//----------------------------------------------------------------------------//
//            Copyright 2018 Rieckermann Engineering Operations               //
//----------------------------------------------------------------------------//
// Class:       fbTC1                                                         //
// Description:                                                               //
// Cooling only temperature controller.                                       //
//----------------------------------------------------------------------------//
// Revision history:                                                          //
// Rev By               Date        CC        Note                            //
// 2.0 David Paspa      24-Apr-2018 NA        Reboot for S7-1500.             //
// 0.7 Gerald Kontriner 09-Oct-2009 CC-09/016 MON_MISMATCH Logic.             //
// 0.6 Khairul Basar    06-Oct-2009 CC-09/016 PID HLM,LLM reversed for cool.  //
// 0.5 Khairul Basar    17-Sep-2009 CC-09/016 OUT_CMD as Command to MOD1 added//
// 0.4 Khairul Basar    16-Sep-2009 CC-09/016 Duplicate Auto/man parameters   //
//                                            deleted auto/manual both now    //
//                                            using same parameters.          //
// 0.3 Khairul Basar    11-Sep-2009 CC-09/016 Manual setpoint, Non PID        //
//                                            selection parameters added &    //
//                                            programmed..                    //
// 0.2 Khairul Basar    03-Sep-2009 CC-09/016 State enable/disable code added //
//                                            NTERLOCK is changed from        //
//                                            IN_OUT to OUT & program safe    //
//                                            state for Interlock.            //
//                                            CMD_AUTO/MAN & DEV_STATE.       //
//                                            paramters are added & programed.//
// 0.1 Khairul Basar    03-Aug-2009           Initial design.                 //
//----------------------------------------------------------------------------//
FUNCTION_BLOCK "fbTC1"
TITLE = TC1 : Vesel cooling only temperature controller
{ S7_Optimized_Access := 'TRUE' }
AUTHOR : REO
NAME : fbTC1
VERSION : 2.0

//----------------------------------------------------------------------------//
// Declare interface and variables:                                           //
//----------------------------------------------------------------------------//
VAR
    p : "udtTC1";            // Block data interface
    PID1 {ReadalPartName := 'CONT_C'; LibVersion := '1.0'} : CONT_C;
END_VAR

VAR_TEMP
    cmdEnable : Bool;
    cmdDisable : Bool;
    tSetpoint : Real;
    tManual_Not_PID : Bool;
END_VAR

BEGIN
NETWORK
TITLE = Check if the TCV is not in AUTO and REMOTE
    //------------------------------------------------------------------------//
    // INTERLOCK   INTERLOCK   INTERLOCK   INTERLOCK   INTERLOCK   INTERLOCK  //
    // INTERLOCK   INTERLOCK   INTERLOCK   INTERLOCK   INTERLOCK   INTERLOCK  //
    //                                                                        //
    // Check if the TCV cannot be controlled if not in AUTO:                  //
    //------------------------------------------------------------------------//
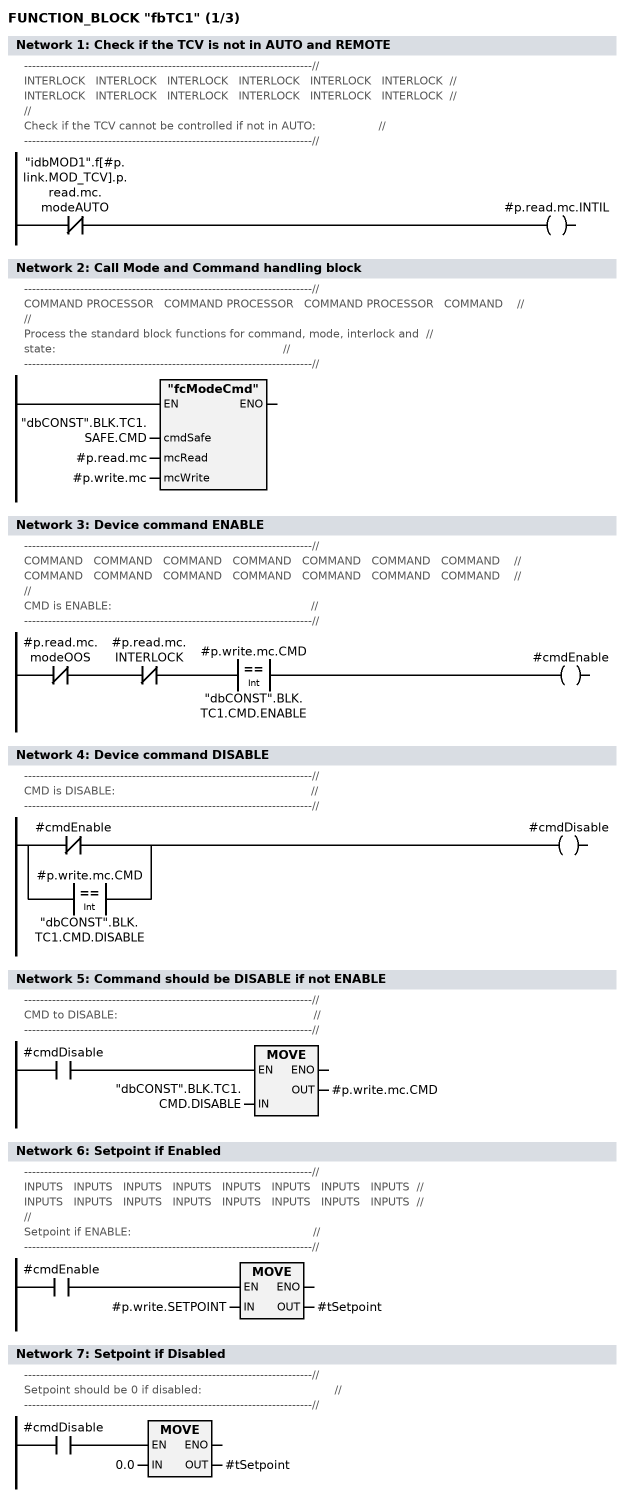
    AN "idbMOD1".f[#p.link.MOD_TCV].p.read.mc.modeAUTO;
    = #p.read.mc.INTIL;

NETWORK
TITLE = Call Mode and Command handling block
    //------------------------------------------------------------------------//
    // COMMAND PROCESSOR   COMMAND PROCESSOR   COMMAND PROCESSOR   COMMAND    //
    //                                                                        //
    // Process the standard block functions for command, mode, interlock and  //
    // state:                                                                 //
    //------------------------------------------------------------------------//
    CALL "fcModeCmd"
    (   cmdSafe              := "dbCONST".BLK.TC1.SAFE.CMD ,
        mcRead               := #p.read.mc ,
        mcWrite              := #p.write.mc
    );

NETWORK
TITLE = Device command ENABLE
    //------------------------------------------------------------------------//
    // COMMAND   COMMAND   COMMAND   COMMAND   COMMAND   COMMAND   COMMAND    //
    // COMMAND   COMMAND   COMMAND   COMMAND   COMMAND   COMMAND   COMMAND    //
    //                                                                        //
    // CMD is ENABLE:                                                         //
    //------------------------------------------------------------------------//
    AN #p.read.mc.modeOOS;
    AN #p.read.mc.INTERLOCK;
    A(;
    L #p.write.mc.CMD;
    L "dbCONST".BLK.TC1.CMD.ENABLE;
    ==I;
    );
    = #cmdEnable;

NETWORK
TITLE = Device command DISABLE
    //------------------------------------------------------------------------//
    // CMD is DISABLE:                                                        //
    //------------------------------------------------------------------------//
    ON #cmdEnable;
    O(;
    L #p.write.mc.CMD;
    L "dbCONST".BLK.TC1.CMD.DISABLE;
    ==I;
    );
    = #cmdDisable;

NETWORK
TITLE = Command should be DISABLE if not ENABLE
    //------------------------------------------------------------------------//
    // CMD to DISABLE:                                                        //
    //------------------------------------------------------------------------//
    A #cmdDisable;
    JCN _a;
    L "dbCONST".BLK.TC1.CMD.DISABLE;
    T #p.write.mc.CMD;
_a:   NOP 0;

NETWORK
TITLE = Setpoint if Enabled
    //------------------------------------------------------------------------//
    // INPUTS   INPUTS   INPUTS   INPUTS   INPUTS   INPUTS   INPUTS   INPUTS  //
    // INPUTS   INPUTS   INPUTS   INPUTS   INPUTS   INPUTS   INPUTS   INPUTS  //
    //                                                                        //
    // Setpoint if ENABLE:                                                    //
    //------------------------------------------------------------------------//
    A #cmdEnable;
    JCN _b;
    L #p.write.SETPOINT;
    T #tSetpoint;
_b:   NOP 0;

NETWORK
TITLE = Setpoint if Disabled
    //------------------------------------------------------------------------//
    // Setpoint should be 0 if disabled:                                      //
    //------------------------------------------------------------------------//
    A #cmdDisable;
    JCN _c;
    L 0.0;
    T #tSetpoint;
_c:   NOP 0;

NETWORK
TITLE = PID in manual if disabled or manual flag set
    //------------------------------------------------------------------------//
    // OUTPUTS   OUTPUTS   OUTPUTS   OUTPUTS   OUTPUTS   OUTPUTS   OUTPUTS    //
    // OUTPUTS   OUTPUTS   OUTPUTS   OUTPUTS   OUTPUTS   OUTPUTS   OUTPUTS    //
    //                                                                        //
    // PID in manual mode if requested:                                       //
    //------------------------------------------------------------------------//
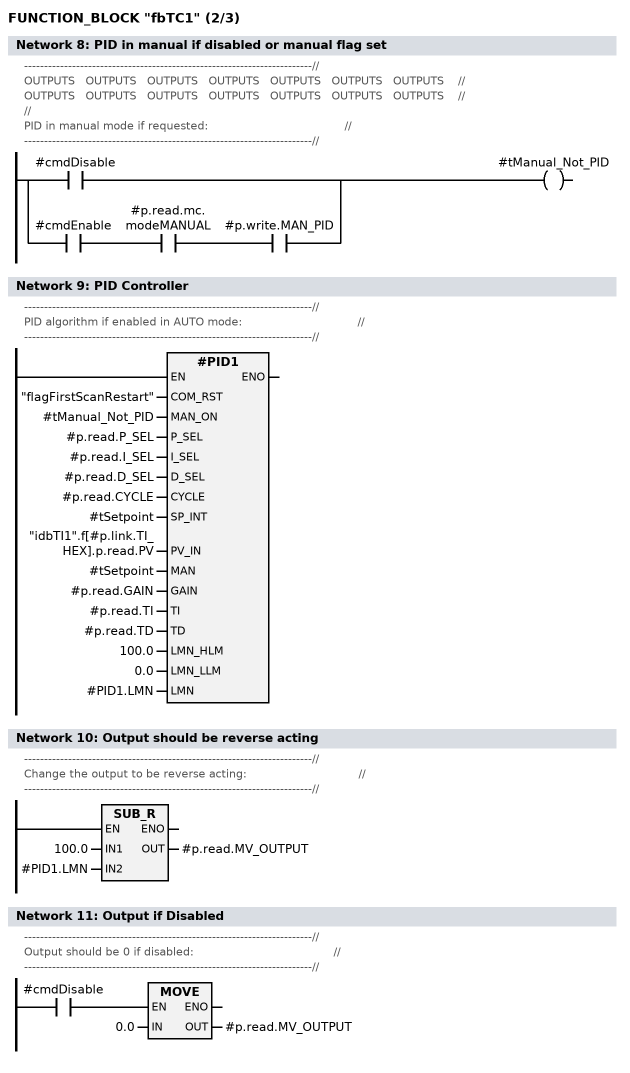
    O #cmdDisable;
    O(;
    A #cmdEnable;
    A #p.read.mc.modeMANUAL;
    A #p.write.MAN_PID;
    );
    = #tManual_Not_PID;

NETWORK
TITLE = PID Controller
    //------------------------------------------------------------------------//
    // PID algorithm if enabled in AUTO mode:                                 //
    //------------------------------------------------------------------------//
    CALL #PID1
    (   COM_RST              := "flagFirstScanRestart" ,
        MAN_ON               := #tManual_Not_PID ,
        P_SEL                := #p.read.P_SEL ,
        I_SEL                := #p.read.I_SEL ,
        D_SEL                := #p.read.D_SEL ,
        CYCLE                := #p.read.CYCLE ,
        SP_INT               := #tSetpoint ,
        PV_IN                := "idbTI1".f[#p.link.TI_HEX].p.read.PV ,
        MAN                  := #tSetpoint ,
        GAIN                 := #p.read.GAIN ,
        TI                   := #p.read.TI ,
        TD                   := #p.read.TD ,
        LMN_HLM              := 100.0 ,
        LMN_LLM              := 0.0 ,
        LMN                  := #PID1.LMN
    );

NETWORK
TITLE = Output should be reverse acting
    //------------------------------------------------------------------------//
    // Change the output to be reverse acting:                                //
    //------------------------------------------------------------------------//
    L 100.0;
    L #PID1.LMN;
    -R;
    T #p.read.MV_OUTPUT;

NETWORK
TITLE = Output if Disabled
    //------------------------------------------------------------------------//
    // Output should be 0 if disabled:                                        //
    //------------------------------------------------------------------------//
    A #cmdDisable;
    JCN _d;
    L 0.0;
    T #p.read.MV_OUTPUT;
_d:   NOP 0;

NETWORK
TITLE = Transfer PID output to MOD1 TC Valve REMOTE setpoint
    //------------------------------------------------------------------------//
    // Write the PID controller output to the temperature control valve (TCV) //
    // remote position setpoint:                                              //
    //------------------------------------------------------------------------//
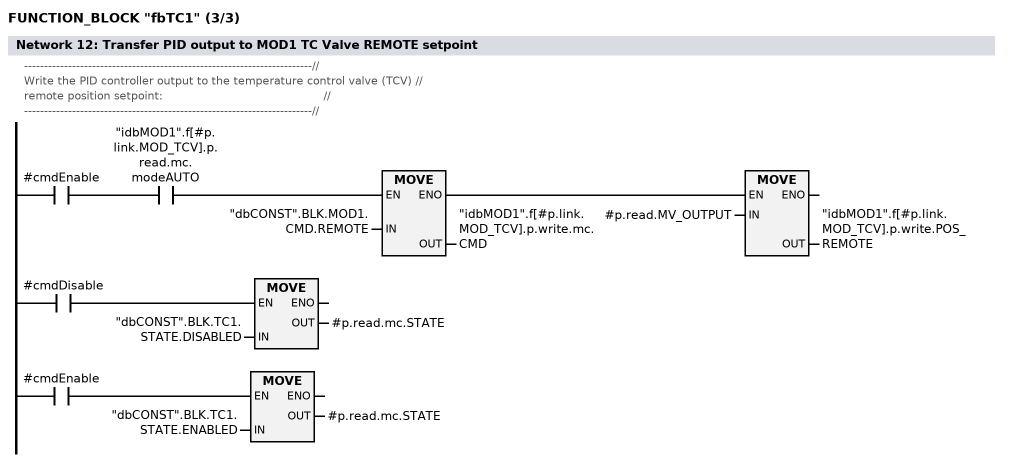
    A #cmdEnable;
    A "idbMOD1".f[#p.link.MOD_TCV].p.read.mc.modeAUTO;
    JCN _notMODAuto;
    L "dbCONST".BLK.MOD1.CMD.REMOTE;
    T "idbMOD1".f[#p.link.MOD_TCV].p.write.mc.CMD;
    L #p.read.MV_OUTPUT;
    T "idbMOD1".f[#p.link.MOD_TCV].p.write.POS_REMOTE;
_notMODAuto:   NOP 0;

    //------------------------------------------------------------------------//
    // STATE   STATE   STATE   STATE   STATE   STATE   STATE   STATE   STATE  //
    // STATE   STATE   STATE   STATE   STATE   STATE   STATE   STATE   STATE  //
    //                                                                        //
    // DISABLED if commanded or any problem or OOS:                           //
    //------------------------------------------------------------------------//
    A #cmdDisable;
    JCN _e;
    L "dbCONST".BLK.TC1.STATE.DISABLED;
    T #p.read.mc.STATE;
_e:   NOP 0;

    //------------------------------------------------------------------------//
    // ENABLED if commanded and no problem:                                   //
    //------------------------------------------------------------------------//
    A #cmdEnable;
    JCN _f;
    L "dbCONST".BLK.TC1.STATE.ENABLED;
    T #p.read.mc.STATE;
_f:   NOP 0;
END_FUNCTION_BLOCK
